Universal Robots PolyScope program: path_offset_sine_weave_UR10_text.urp

Program path_offset_sine_weave_UR10 (installation=path_offset_sine_weave_UR10 directory=/home/ask/git/polyscope/staging/programs createdIn=5.5.0.0 lastSavedIn=5.5.0.0 robotSerialNumber=20175099999)
Calibrated DH parameters: a=[0, -0.6127, -0.57155, 0, 0, 0]; d=[0.1807, 0, 0, 0.17415, 0.11985, 0.11655]; alpha=[1.570796, 0, 0, 1.570796, -1.570796, 0]; deltaTheta=[0, 0, 0, 0, 0, 0]
Robot Program (runOnlyOnce=true)
  MoveP speed 8 mm/s, acceleration 1200 mm/s^2 (blendRadius=0.025 useActiveTCP=true) feature=Base
    Waypoint start_pos: TCP in base x=-200 y=-700 z=100 mm, rx=0 ry=3.1168 rz=0 rad; joints [-92.339, -119.741, -120.476, -29.841, 91.421, -2.34] deg; TCP offset x=0 y=0 z=0 mm, rx=0 ry=0 rz=0 rad
    Waypoint end_pos: TCP in base x=100 y=-700 z=100 mm, rx=0 ry=3.1168 rz=0 rad; joints [-67.836, -118.644, -123.011, -27.808, 91.317, 22.17] deg; TCP offset x=0 y=0 z=0 mm, rx=0 ry=0 rz=0 rad
Thread Thread_1 (runOnlyOnce=false)
  Folder setup
    ctrl_frequency := 500.0
    weave_frequency := 3.0
    amplitude := 0.006
    cycle_duration := ctrl_frequency / weave_frequency
    pi := 3.14159
  Folder enable
    offset := [0.0, 0.0, 0.0, 0.0, 0.0, 0.0]
    i := 0
    Script: path_offset_enable()
    alpha := 0.27
    Script: path_offset_set_alpha_filter(alpha)
  Folder weave
    Loop Forever
      Script: offset[1]=sin((i / cycle_duration) * 2.0 * pi) * amplitude
      Script: path_offset_set(offset, 2)
      i := i+1
      Script: sync()
